{attribute 'qualified_only'}
VAR_GLOBAL CONSTANT
	MAX_NUMBER_IMAGES_2_VIDEO : UDINT := 200;
	MAX_PERCENT_ROUTER_MEM_FOR_BUFFER : UDINT := 50;
	ADS_PORT_FOR_IMAGE_TO_VIDEO		  : UINT  := 26129;
	LARGE_ROUTER_MEMORY				  : UINT  := 4096;
END_VAR

(* stored: Version 1.1.0.1
   GVL Parameters_EventVideoPlayback: Id {56c9dfe6-e032-0b0f-1edc-689100bf16fe}, ParameterList True *)
